// TIA Portal V16 export
// export: Created 2022-09-01T13:58:53.9075571Z, ExportSetting WithDefaults, DisplayName Totally Integrated Automation Portal, DisplayVersion V16, DisplayName TIA Portal Version Control Interface, DisplayVersion V16, DisplayName TIA Portal Openness, DisplayVersion V16, DisplayName STEP 7 Professional, DisplayVersion V16, DisplayName STEP 7 Safety, DisplayVersion V16, DisplayName WinCC Advanced, DisplayVersion V16
DATA_BLOCK "Dados_Ciclo"   // DB7
{ S7_Optimized_Access := 'TRUE' }
VERSION : 0.1
// stored: AutoNumber true, IsOnlyStoredInLoadMemory false, IsRetainMemResEnabled false, IsWriteProtectedInAS false, MemoryReserve 100
   VAR
      HOLD_ETAPA_1 : Bool;
   END_VAR
   VAR RETAIN
      FILTRO1_EM_CICLO : Bool;
      FILTRO2_EM_CICLO : Bool;
      FECHO_FILT_1 : Bool;
      FECHO_FILT_2 : Bool;
      ETAPA_ANTERIOR : Int := 1;
   END_VAR
   VAR
      ETAPA_N : Bool;
      POS_EVS_FILT_1 : String;
      POS_EVS_FILT_2 : String;
      PRESS_SP_FILT_1 : Bool;
      PRESS_SP_FILT_2 : Bool;
   END_VAR
   VAR RETAIN
      STOP_CICLO : Bool;
   END_VAR
   VAR
      AGEND_FILT_1 : Bool;
      AGEND_FILT_2 : Bool;
   END_VAR
   VAR RETAIN
      HORA_INIC_FILT_1 : USInt;
      MIN_INIC_FILT_1 : USInt;
      HORA_INIC_FILT_2 : USInt;
      MIN_INIC_FILT_2 : USInt;
      ENABLE_AGEND_FILT_1 : Bool;
      ENABLE_AGEND_FILT_2 : Bool;
   END_VAR
   VAR
      PRESSÃO_FILT1 : Real;
      PRESSÃO_FILT2 : Real;
   END_VAR
BEGIN
END_DATA_BLOCK
